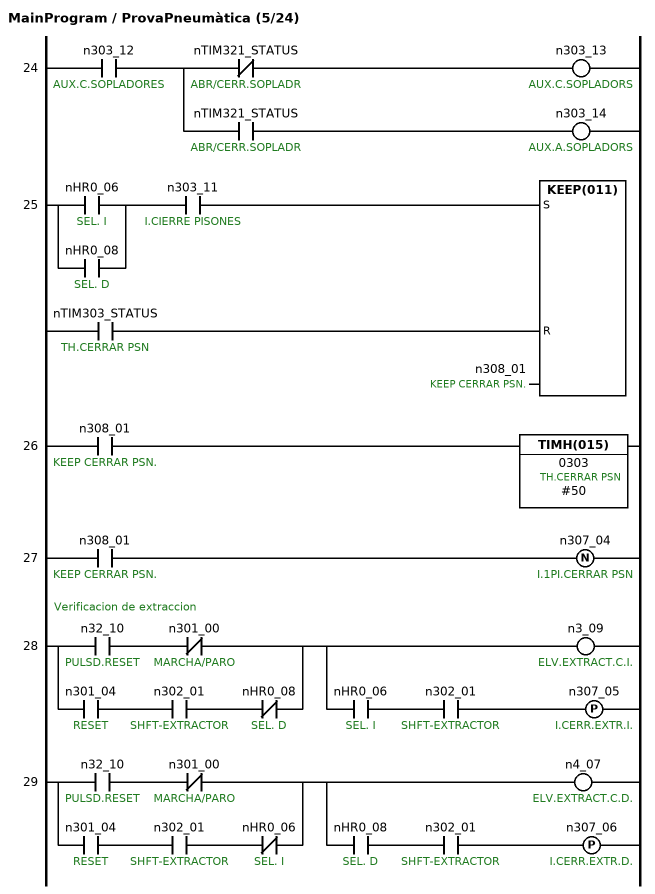
; [picture p96: MainProgram / ProvaPneumàtica, rungs 24-29]
; rung 24
LD n303_12  ; AUX.C.SOPLADORES
OUT TR0
ANDNOT nTIM321_STATUS  ; ABR/CERR.SOPLADR
OUT n303_13  ; AUX.C.SOPLADORS
LD TR0
AND nTIM321_STATUS  ; ABR/CERR.SOPLADR
OUT n303_14  ; AUX.A.SOPLADORS
; rung 25
LD nHR0_06  ; SEL. I
OR nHR0_08  ; SEL. D
AND n303_11  ; I.CIERRE PISONES
LD nTIM303_STATUS  ; TH.CERRAR PSN
KEEP(011) n308_01  ; KEEP CERRAR PSN.
; rung 26
LD n308_01  ; KEEP CERRAR PSN.
TIMH(015) 0303 #50  ; TH.CERRAR PSN
; rung 27
LD n308_01  ; KEEP CERRAR PSN.
DIFD(014) n307_04  ; I.1PI.CERRAR PSN
; rung 28: Verificacion de extraccion
LD n32_10  ; PULSD.RESET
ANDNOT n301_00  ; MARCHA/PARO
LD n301_04  ; RESET
AND n302_01  ; SHFT-EXTRACTOR
ANDNOT nHR0_08  ; SEL. D
ORLD
OUT n3_09  ; ELV.EXTRACT.C.I.
AND nHR0_06  ; SEL. I
AND n302_01  ; SHFT-EXTRACTOR
DIFU(013) n307_05  ; I.CERR.EXTR.I.
; rung 29
LD n32_10  ; PULSD.RESET
ANDNOT n301_00  ; MARCHA/PARO
LD n301_04  ; RESET
AND n302_01  ; SHFT-EXTRACTOR
ANDNOT nHR0_06  ; SEL. I
ORLD
OUT n4_07  ; ELV.EXTRACT.C.D.
AND nHR0_08  ; SEL. D
AND n302_01  ; SHFT-EXTRACTOR
DIFU(013) n307_06  ; I.CERR.EXTR.D.

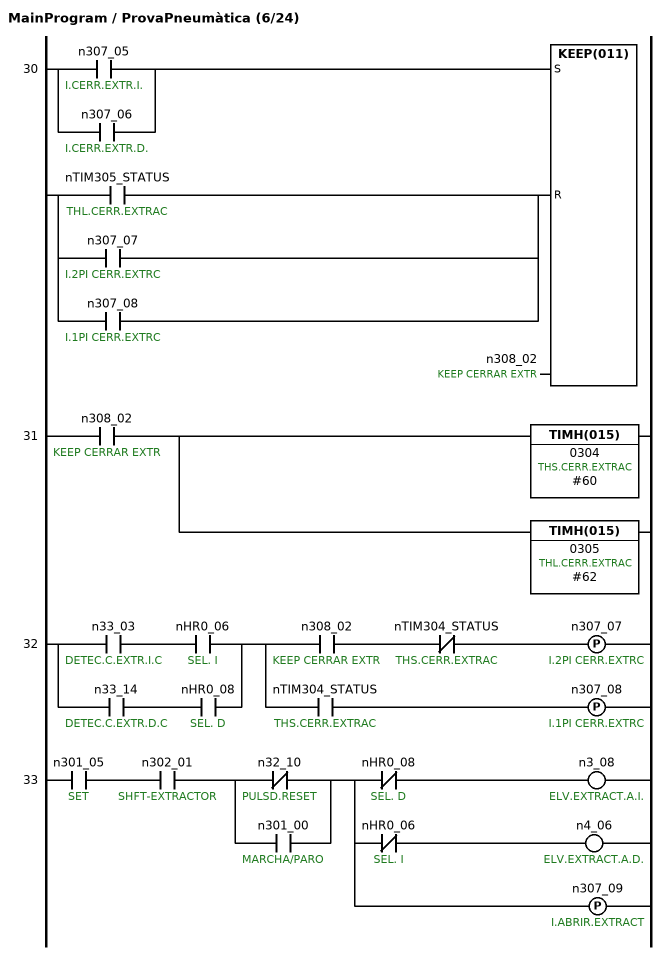
; rung 30
LD n307_05  ; I.CERR.EXTR.I.
OR n307_06  ; I.CERR.EXTR.D.
LD nTIM305_STATUS  ; THL.CERR.EXTRAC
OR n307_07  ; I.2PI CERR.EXTRC
OR n307_08  ; I.1PI CERR.EXTRC
KEEP(011) n308_02  ; KEEP CERRAR EXTR
; rung 31
LD n308_02  ; KEEP CERRAR EXTR
TIMH(015) 0304 #60  ; THS.CERR.EXTRAC
TIMH(015) 0305 #62  ; THL.CERR.EXTRAC
; rung 32
LD n33_03  ; DETEC.C.EXTR.I.C
AND nHR0_06  ; SEL. I
LD n33_14  ; DETEC.C.EXTR.D.C
AND nHR0_08  ; SEL. D
ORLD
OUT TR0
AND n308_02  ; KEEP CERRAR EXTR
ANDNOT nTIM304_STATUS  ; THS.CERR.EXTRAC
DIFU(013) n307_07  ; I.2PI CERR.EXTRC
LD TR0
AND nTIM304_STATUS  ; THS.CERR.EXTRAC
DIFU(013) n307_08  ; I.1PI CERR.EXTRC
; rung 33
LD n301_05  ; SET
AND n302_01  ; SHFT-EXTRACTOR
LDNOT n32_10  ; PULSD.RESET
OR n301_00  ; MARCHA/PARO
ANDLD
OUT TR0
ANDNOT nHR0_08  ; SEL. D
OUT n3_08  ; ELV.EXTRACT.A.I.
LD TR0
ANDNOT nHR0_06  ; SEL. I
OUT n4_06  ; ELV.EXTRACT.A.D.
LD TR0
DIFU(013) n307_09  ; I.ABRIR.EXTRACT

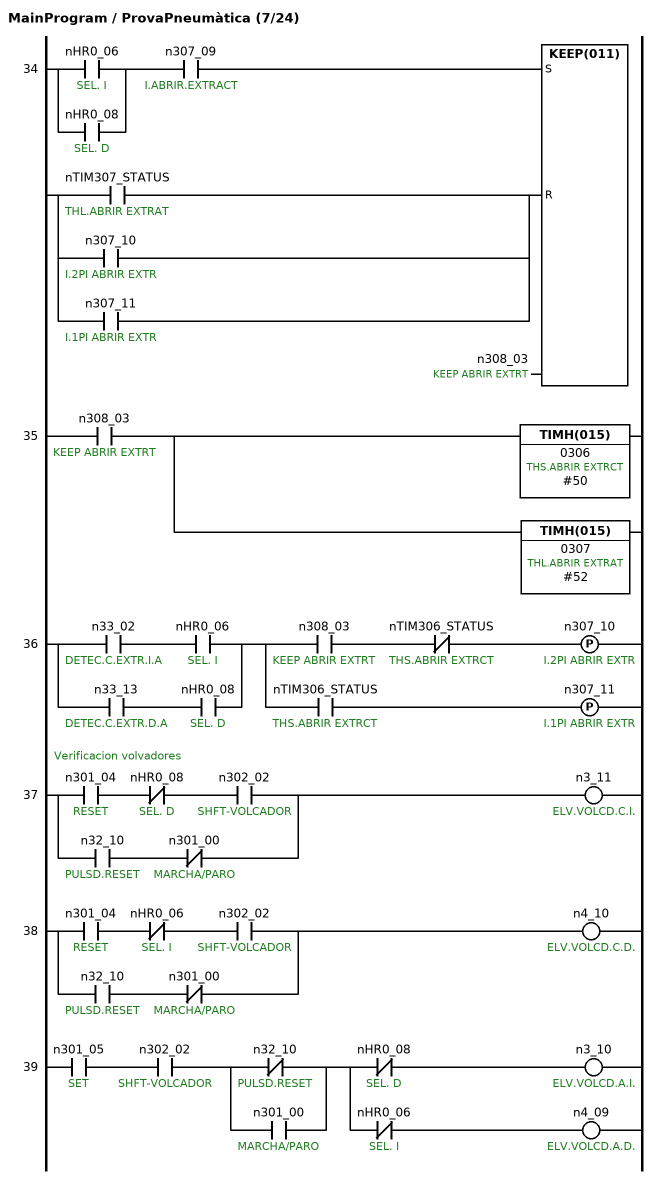
; rung 34
LD nHR0_06  ; SEL. I
OR nHR0_08  ; SEL. D
AND n307_09  ; I.ABRIR.EXTRACT
LD nTIM307_STATUS  ; THL.ABRIR EXTRAT
OR n307_10  ; I.2PI ABRIR EXTR
OR n307_11  ; I.1PI ABRIR EXTR
KEEP(011) n308_03  ; KEEP ABRIR EXTRT
; rung 35
LD n308_03  ; KEEP ABRIR EXTRT
TIMH(015) 0306 #50  ; THS.ABRIR EXTRCT
TIMH(015) 0307 #52  ; THL.ABRIR EXTRAT
; rung 36
LD n33_02  ; DETEC.C.EXTR.I.A
AND nHR0_06  ; SEL. I
LD n33_13  ; DETEC.C.EXTR.D.A
AND nHR0_08  ; SEL. D
ORLD
OUT TR0
AND n308_03  ; KEEP ABRIR EXTRT
ANDNOT nTIM306_STATUS  ; THS.ABRIR EXTRCT
DIFU(013) n307_10  ; I.2PI ABRIR EXTR
LD TR0
AND nTIM306_STATUS  ; THS.ABRIR EXTRCT
DIFU(013) n307_11  ; I.1PI ABRIR EXTR
; rung 37: Verificacion volvadores
LD n301_04  ; RESET
ANDNOT nHR0_08  ; SEL. D
AND n302_02  ; SHFT-VOLCADOR
LD n32_10  ; PULSD.RESET
ANDNOT n301_00  ; MARCHA/PARO
ORLD
OUT n3_11  ; ELV.VOLCD.C.I.
; rung 38
LD n301_04  ; RESET
ANDNOT nHR0_06  ; SEL. I
AND n302_02  ; SHFT-VOLCADOR
LD n32_10  ; PULSD.RESET
ANDNOT n301_00  ; MARCHA/PARO
ORLD
OUT n4_10  ; ELV.VOLCD.C.D.
; rung 39
LD n301_05  ; SET
AND n302_02  ; SHFT-VOLCADOR
LDNOT n32_10  ; PULSD.RESET
OR n301_00  ; MARCHA/PARO
ANDLD
OUT TR0
ANDNOT nHR0_08  ; SEL. D
OUT n3_10  ; ELV.VOLCD.A.I.
LD TR0
ANDNOT nHR0_06  ; SEL. I
OUT n4_09  ; ELV.VOLCD.A.D.

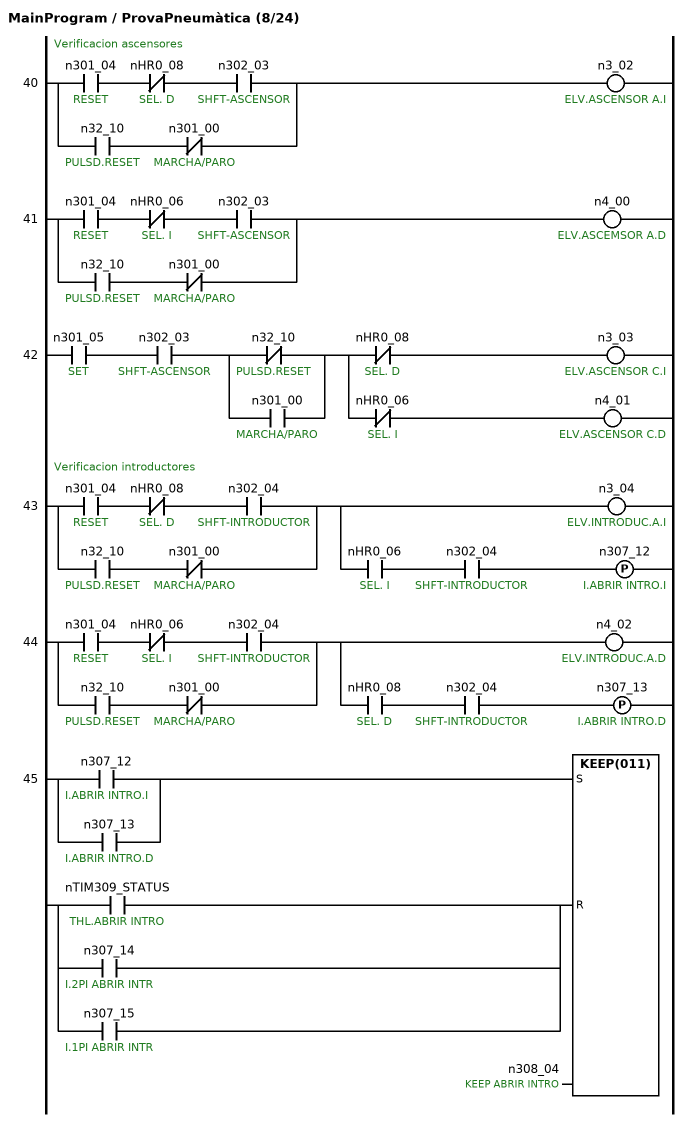
; rung 40: Verificacion ascensores
LD n301_04  ; RESET
ANDNOT nHR0_08  ; SEL. D
AND n302_03  ; SHFT-ASCENSOR
LD n32_10  ; PULSD.RESET
ANDNOT n301_00  ; MARCHA/PARO
ORLD
OUT n3_02  ; ELV.ASCENSOR A.I
; rung 41
LD n301_04  ; RESET
ANDNOT nHR0_06  ; SEL. I
AND n302_03  ; SHFT-ASCENSOR
LD n32_10  ; PULSD.RESET
ANDNOT n301_00  ; MARCHA/PARO
ORLD
OUT n4_00  ; ELV.ASCEMSOR A.D
; rung 42
LD n301_05  ; SET
AND n302_03  ; SHFT-ASCENSOR
LDNOT n32_10  ; PULSD.RESET
OR n301_00  ; MARCHA/PARO
ANDLD
OUT TR0
ANDNOT nHR0_08  ; SEL. D
OUT n3_03  ; ELV.ASCENSOR C.I
LD TR0
ANDNOT nHR0_06  ; SEL. I
OUT n4_01  ; ELV.ASCENSOR C.D
; rung 43: Verificacion introductores
LD n301_04  ; RESET
ANDNOT nHR0_08  ; SEL. D
AND n302_04  ; SHFT-INTRODUCTOR
LD n32_10  ; PULSD.RESET
ANDNOT n301_00  ; MARCHA/PARO
ORLD
OUT n3_04  ; ELV.INTRODUC.A.I
AND nHR0_06  ; SEL. I
AND n302_04  ; SHFT-INTRODUCTOR
DIFU(013) n307_12  ; I.ABRIR INTRO.I
; rung 44
LD n301_04  ; RESET
ANDNOT nHR0_06  ; SEL. I
AND n302_04  ; SHFT-INTRODUCTOR
LD n32_10  ; PULSD.RESET
ANDNOT n301_00  ; MARCHA/PARO
ORLD
OUT n4_02  ; ELV.INTRODUC.A.D
AND nHR0_08  ; SEL. D
AND n302_04  ; SHFT-INTRODUCTOR
DIFU(013) n307_13  ; I.ABRIR INTRO.D
; rung 45
LD n307_12  ; I.ABRIR INTRO.I
OR n307_13  ; I.ABRIR INTRO.D
LD nTIM309_STATUS  ; THL.ABRIR INTRO
OR n307_14  ; I.2PI ABRIR INTR
OR n307_15  ; I.1PI ABRIR INTR
KEEP(011) n308_04  ; KEEP ABRIR INTRO

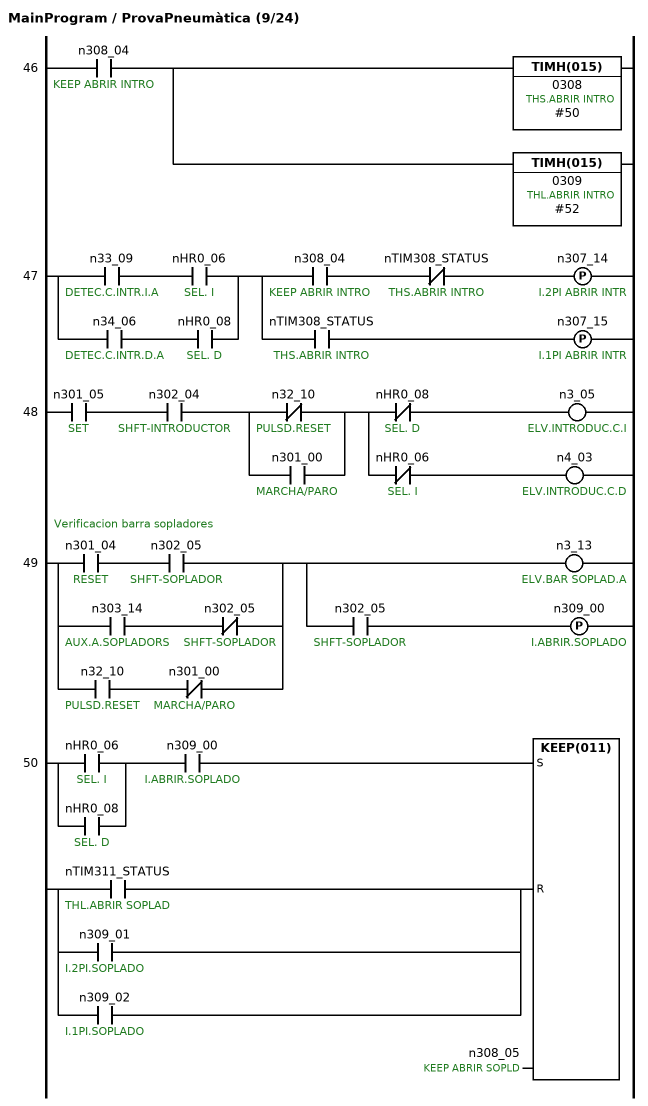
; rung 46
LD n308_04  ; KEEP ABRIR INTRO
TIMH(015) 0308 #50  ; THS.ABRIR INTRO
TIMH(015) 0309 #52  ; THL.ABRIR INTRO
; rung 47
LD n33_09  ; DETEC.C.INTR.I.A
AND nHR0_06  ; SEL. I
LD n34_06  ; DETEC.C.INTR.D.A
AND nHR0_08  ; SEL. D
ORLD
OUT TR0
AND n308_04  ; KEEP ABRIR INTRO
ANDNOT nTIM308_STATUS  ; THS.ABRIR INTRO
DIFU(013) n307_14  ; I.2PI ABRIR INTR
LD TR0
AND nTIM308_STATUS  ; THS.ABRIR INTRO
DIFU(013) n307_15  ; I.1PI ABRIR INTR
; rung 48
LD n301_05  ; SET
AND n302_04  ; SHFT-INTRODUCTOR
LDNOT n32_10  ; PULSD.RESET
OR n301_00  ; MARCHA/PARO
ANDLD
OUT TR0
ANDNOT nHR0_08  ; SEL. D
OUT n3_05  ; ELV.INTRODUC.C.I
LD TR0
ANDNOT nHR0_06  ; SEL. I
OUT n4_03  ; ELV.INTRODUC.C.D
; rung 49: Verificacion barra sopladores
LD n301_04  ; RESET
AND n302_05  ; SHFT-SOPLADOR
LD n303_14  ; AUX.A.SOPLADORS
ANDNOT n302_05  ; SHFT-SOPLADOR
ORLD
LD n32_10  ; PULSD.RESET
ANDNOT n301_00  ; MARCHA/PARO
ORLD
OUT n3_13  ; ELV.BAR SOPLAD.A
AND n302_05  ; SHFT-SOPLADOR
DIFU(013) n309_00  ; I.ABRIR.SOPLADO
; rung 50
LD nHR0_06  ; SEL. I
OR nHR0_08  ; SEL. D
AND n309_00  ; I.ABRIR.SOPLADO
LD nTIM311_STATUS  ; THL.ABRIR SOPLAD
OR n309_01  ; I.2PI.SOPLADO
OR n309_02  ; I.1PI.SOPLADO
KEEP(011) n308_05  ; KEEP ABRIR SOPLD

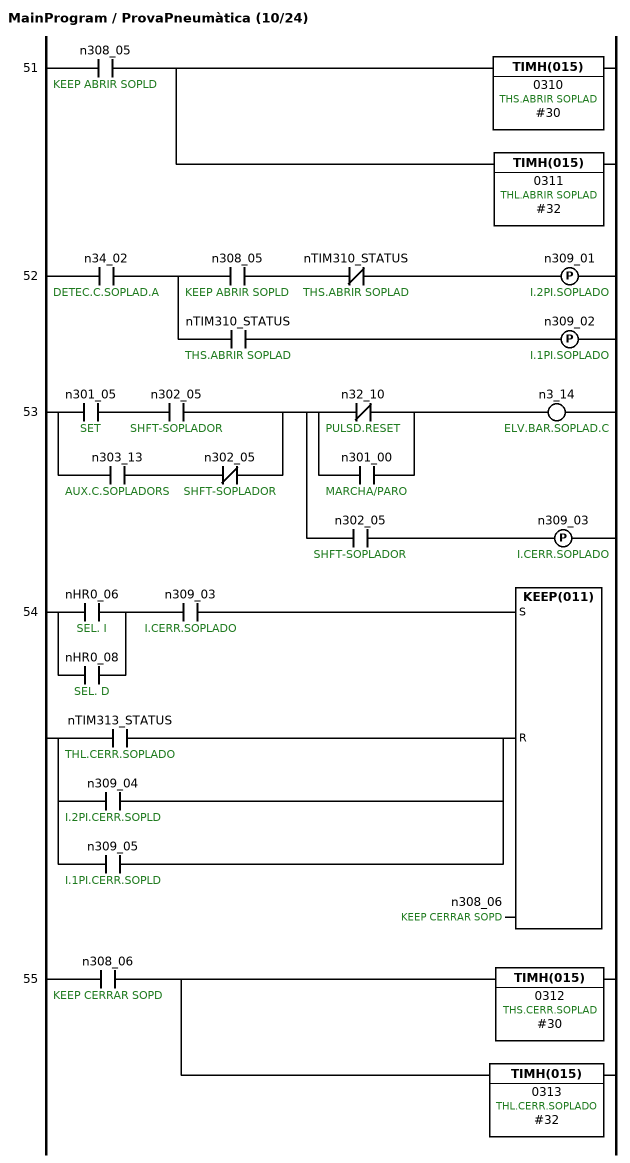
; rung 51
LD n308_05  ; KEEP ABRIR SOPLD
TIMH(015) 0310 #30  ; THS.ABRIR SOPLAD
TIMH(015) 0311 #32  ; THL.ABRIR SOPLAD
; rung 52
LD n34_02  ; DETEC.C.SOPLAD.A
OUT TR0
AND n308_05  ; KEEP ABRIR SOPLD
ANDNOT nTIM310_STATUS  ; THS.ABRIR SOPLAD
DIFU(013) n309_01  ; I.2PI.SOPLADO
LD TR0
AND nTIM310_STATUS  ; THS.ABRIR SOPLAD
DIFU(013) n309_02  ; I.1PI.SOPLADO
; rung 53
LD n301_05  ; SET
AND n302_05  ; SHFT-SOPLADOR
LD n303_13  ; AUX.C.SOPLADORS
ANDNOT n302_05  ; SHFT-SOPLADOR
ORLD
OUT TR0
LDNOT n32_10  ; PULSD.RESET
OR n301_00  ; MARCHA/PARO
ANDLD
OUT n3_14  ; ELV.BAR.SOPLAD.C
LD TR0
AND n302_05  ; SHFT-SOPLADOR
DIFU(013) n309_03  ; I.CERR.SOPLADO
; rung 54
LD nHR0_06  ; SEL. I
OR nHR0_08  ; SEL. D
AND n309_03  ; I.CERR.SOPLADO
LD nTIM313_STATUS  ; THL.CERR.SOPLADO
OR n309_04  ; I.2PI.CERR.SOPLD
OR n309_05  ; I.1PI.CERR.SOPLD
KEEP(011) n308_06  ; KEEP CERRAR SOPD
; rung 55
LD n308_06  ; KEEP CERRAR SOPD
TIMH(015) 0312 #30  ; THS.CERR.SOPLAD
TIMH(015) 0313 #32  ; THL.CERR.SOPLADO

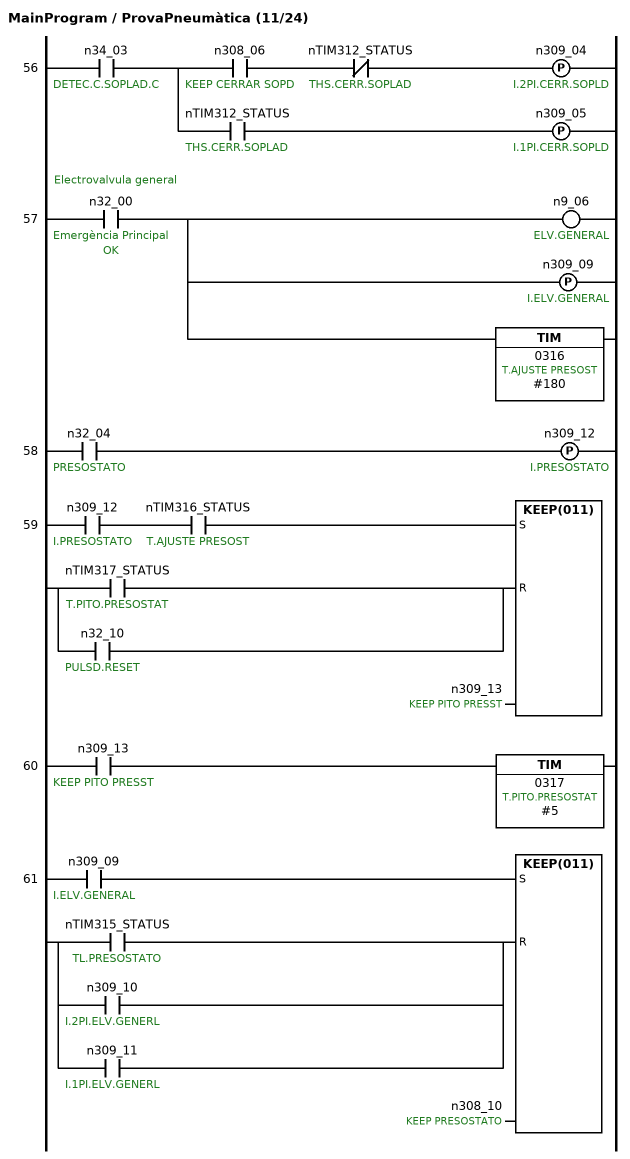
; rung 56
LD n34_03  ; DETEC.C.SOPLAD.C
OUT TR0
AND n308_06  ; KEEP CERRAR SOPD
ANDNOT nTIM312_STATUS  ; THS.CERR.SOPLAD
DIFU(013) n309_04  ; I.2PI.CERR.SOPLD
LD TR0
AND nTIM312_STATUS  ; THS.CERR.SOPLAD
DIFU(013) n309_05  ; I.1PI.CERR.SOPLD
; rung 57: Electrovalvula general
LD n32_00  ; Emergència Principal OK
OUT n9_06  ; ELV.GENERAL
DIFU(013) n309_09  ; I.ELV.GENERAL
TIM 0316 #180  ; T.AJUSTE PRESOST
; rung 58
LD n32_04  ; PRESOSTATO
DIFU(013) n309_12  ; I.PRESOSTATO
; rung 59
LD n309_12  ; I.PRESOSTATO
AND nTIM316_STATUS  ; T.AJUSTE PRESOST
LD nTIM317_STATUS  ; T.PITO.PRESOSTAT
OR n32_10  ; PULSD.RESET
KEEP(011) n309_13  ; KEEP PITO PRESST
; rung 60
LD n309_13  ; KEEP PITO PRESST
TIM 0317 #5  ; T.PITO.PRESOSTAT
; rung 61
LD n309_09  ; I.ELV.GENERAL
LD nTIM315_STATUS  ; TL.PRESOSTATO
OR n309_10  ; I.2PI.ELV.GENERL
OR n309_11  ; I.1PI.ELV.GENERL
KEEP(011) n308_10  ; KEEP PRESOSTATO

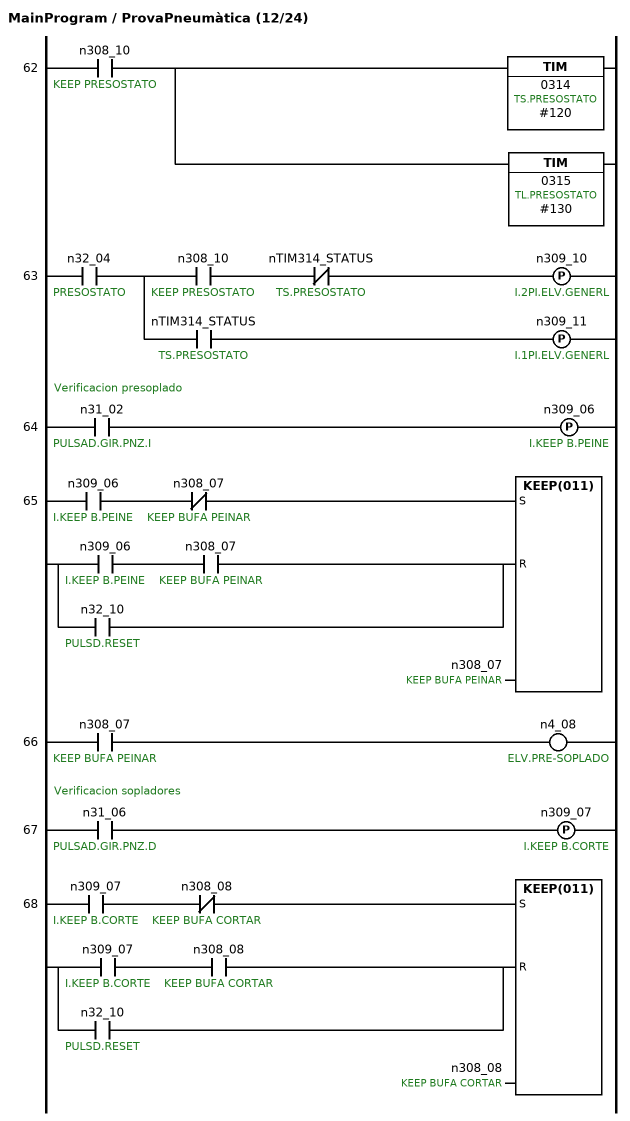
; rung 62
LD n308_10  ; KEEP PRESOSTATO
TIM 0314 #120  ; TS.PRESOSTATO
TIM 0315 #130  ; TL.PRESOSTATO
; rung 63
LD n32_04  ; PRESOSTATO
OUT TR0
AND n308_10  ; KEEP PRESOSTATO
ANDNOT nTIM314_STATUS  ; TS.PRESOSTATO
DIFU(013) n309_10  ; I.2PI.ELV.GENERL
LD TR0
AND nTIM314_STATUS  ; TS.PRESOSTATO
DIFU(013) n309_11  ; I.1PI.ELV.GENERL
; rung 64: Verificacion presoplado
LD n31_02  ; PULSAD.GIR.PNZ.I
DIFU(013) n309_06  ; I.KEEP B.PEINE
; rung 65
LD n309_06  ; I.KEEP B.PEINE
ANDNOT n308_07  ; KEEP BUFA PEINAR
LD n309_06  ; I.KEEP B.PEINE
AND n308_07  ; KEEP BUFA PEINAR
OR n32_10  ; PULSD.RESET
KEEP(011) n308_07  ; KEEP BUFA PEINAR
; rung 66
LD n308_07  ; KEEP BUFA PEINAR
OUT n4_08  ; ELV.PRE-SOPLADO
; rung 67: Verificacion sopladores
LD n31_06  ; PULSAD.GIR.PNZ.D
DIFU(013) n309_07  ; I.KEEP B.CORTE
; rung 68
LD n309_07  ; I.KEEP B.CORTE
ANDNOT n308_08  ; KEEP BUFA CORTAR
LD n309_07  ; I.KEEP B.CORTE
AND n308_08  ; KEEP BUFA CORTAR
OR n32_10  ; PULSD.RESET
KEEP(011) n308_08  ; KEEP BUFA CORTAR

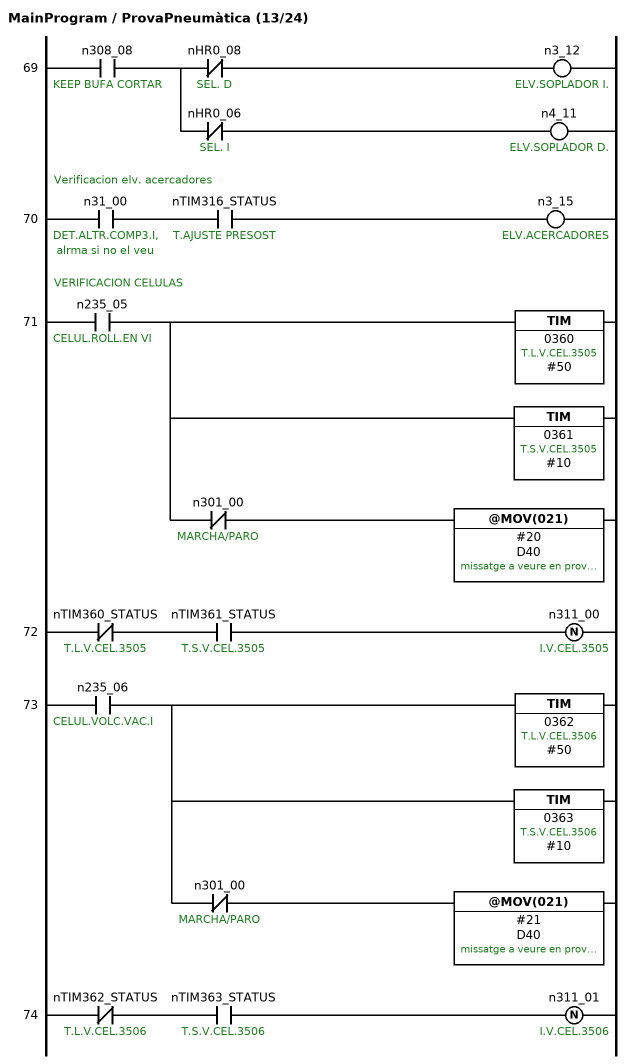
; rung 69
LD n308_08  ; KEEP BUFA CORTAR
OUT TR0
ANDNOT nHR0_08  ; SEL. D
OUT n3_12  ; ELV.SOPLADOR I.
LD TR0
ANDNOT nHR0_06  ; SEL. I
OUT n4_11  ; ELV.SOPLADOR D.
; rung 70: Verificacion elv. acercadores
LD n31_00  ; DET.ALTR.COMP3.I, alrma si no el veu
AND nTIM316_STATUS  ; T.AJUSTE PRESOST
OUT n3_15  ; ELV.ACERCADORES
; rung 71: VERIFICACION CELULAS
LD n235_05  ; CELUL.ROLL.EN VI
TIM 0360 #50  ; T.L.V.CEL.3505
TIM 0361 #10  ; T.S.V.CEL.3505
ANDNOT n301_00  ; MARCHA/PARO
@MOV(021) #20 D40  ; missatge a veure en prova pneumàtica
; rung 72
LDNOT nTIM360_STATUS  ; T.L.V.CEL.3505
AND nTIM361_STATUS  ; T.S.V.CEL.3505
DIFD(014) n311_00  ; I.V.CEL.3505
; rung 73
LD n235_06  ; CELUL.VOLC.VAC.I
TIM 0362 #50  ; T.L.V.CEL.3506
TIM 0363 #10  ; T.S.V.CEL.3506
ANDNOT n301_00  ; MARCHA/PARO
@MOV(021) #21 D40  ; missatge a veure en prova pneumàtica
; rung 74
LDNOT nTIM362_STATUS  ; T.L.V.CEL.3506
AND nTIM363_STATUS  ; T.S.V.CEL.3506
DIFD(014) n311_01  ; I.V.CEL.3506

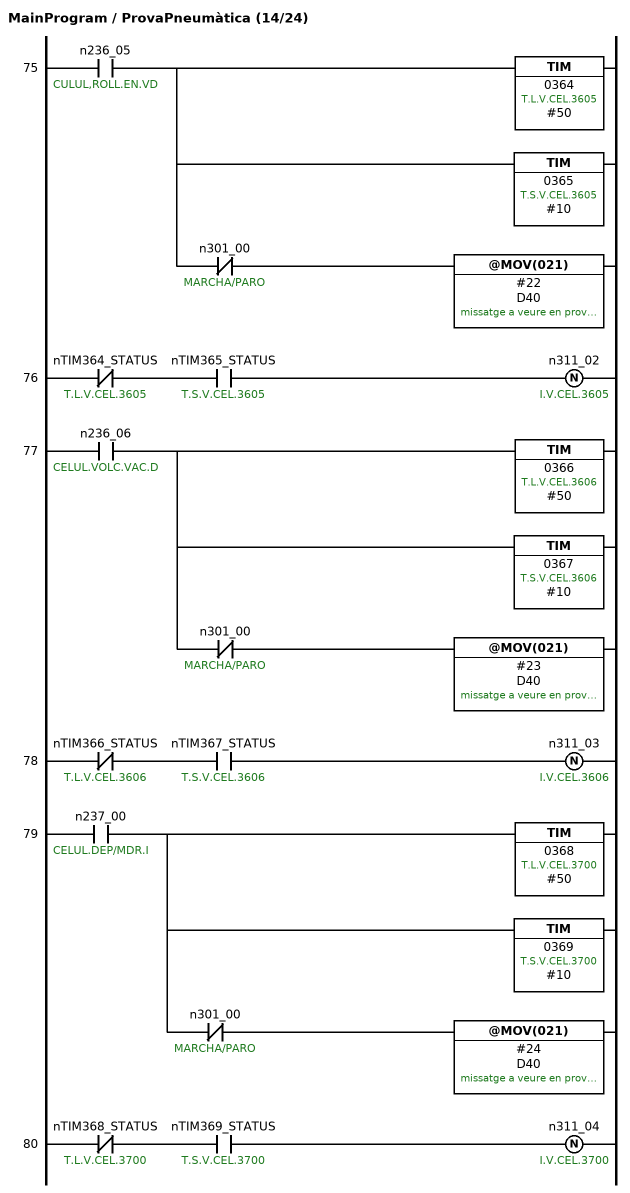
; rung 75
LD n236_05  ; CULUL,ROLL.EN.VD
TIM 0364 #50  ; T.L.V.CEL.3605
TIM 0365 #10  ; T.S.V.CEL.3605
ANDNOT n301_00  ; MARCHA/PARO
@MOV(021) #22 D40  ; missatge a veure en prova pneumàtica
; rung 76
LDNOT nTIM364_STATUS  ; T.L.V.CEL.3605
AND nTIM365_STATUS  ; T.S.V.CEL.3605
DIFD(014) n311_02  ; I.V.CEL.3605
; rung 77
LD n236_06  ; CELUL.VOLC.VAC.D
TIM 0366 #50  ; T.L.V.CEL.3606
TIM 0367 #10  ; T.S.V.CEL.3606
ANDNOT n301_00  ; MARCHA/PARO
@MOV(021) #23 D40  ; missatge a veure en prova pneumàtica
; rung 78
LDNOT nTIM366_STATUS  ; T.L.V.CEL.3606
AND nTIM367_STATUS  ; T.S.V.CEL.3606
DIFD(014) n311_03  ; I.V.CEL.3606
; rung 79
LD n237_00  ; CELUL.DEP/MDR.I
TIM 0368 #50  ; T.L.V.CEL.3700
TIM 0369 #10  ; T.S.V.CEL.3700
ANDNOT n301_00  ; MARCHA/PARO
@MOV(021) #24 D40  ; missatge a veure en prova pneumàtica
; rung 80
LDNOT nTIM368_STATUS  ; T.L.V.CEL.3700
AND nTIM369_STATUS  ; T.S.V.CEL.3700
DIFD(014) n311_04  ; I.V.CEL.3700

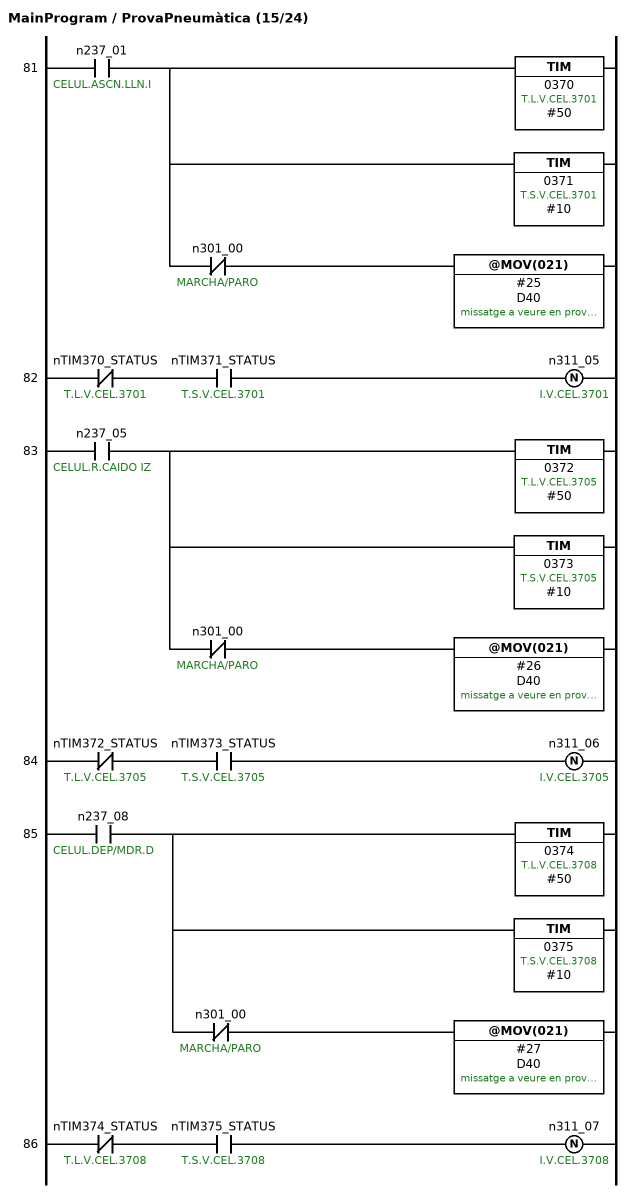
; rung 81
LD n237_01  ; CELUL.ASCN.LLN.I
TIM 0370 #50  ; T.L.V.CEL.3701
TIM 0371 #10  ; T.S.V.CEL.3701
ANDNOT n301_00  ; MARCHA/PARO
@MOV(021) #25 D40  ; missatge a veure en prova pneumàtica
; rung 82
LDNOT nTIM370_STATUS  ; T.L.V.CEL.3701
AND nTIM371_STATUS  ; T.S.V.CEL.3701
DIFD(014) n311_05  ; I.V.CEL.3701
; rung 83
LD n237_05  ; CELUL.R.CAIDO IZ
TIM 0372 #50  ; T.L.V.CEL.3705
TIM 0373 #10  ; T.S.V.CEL.3705
ANDNOT n301_00  ; MARCHA/PARO
@MOV(021) #26 D40  ; missatge a veure en prova pneumàtica
; rung 84
LDNOT nTIM372_STATUS  ; T.L.V.CEL.3705
AND nTIM373_STATUS  ; T.S.V.CEL.3705
DIFD(014) n311_06  ; I.V.CEL.3705
; rung 85
LD n237_08  ; CELUL.DEP/MDR.D
TIM 0374 #50  ; T.L.V.CEL.3708
TIM 0375 #10  ; T.S.V.CEL.3708
ANDNOT n301_00  ; MARCHA/PARO
@MOV(021) #27 D40  ; missatge a veure en prova pneumàtica
; rung 86
LDNOT nTIM374_STATUS  ; T.L.V.CEL.3708
AND nTIM375_STATUS  ; T.S.V.CEL.3708
DIFD(014) n311_07  ; I.V.CEL.3708

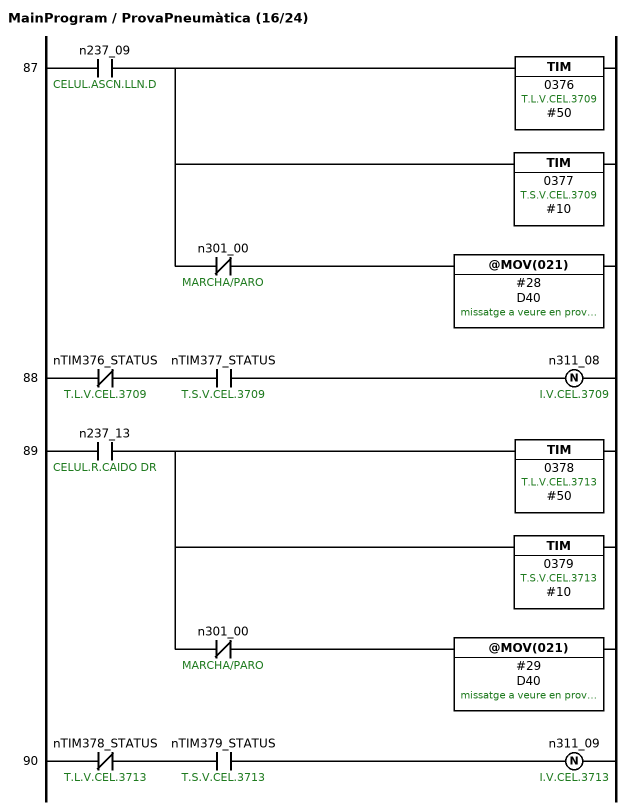
; rung 87
LD n237_09  ; CELUL.ASCN.LLN.D
TIM 0376 #50  ; T.L.V.CEL.3709
TIM 0377 #10  ; T.S.V.CEL.3709
ANDNOT n301_00  ; MARCHA/PARO
@MOV(021) #28 D40  ; missatge a veure en prova pneumàtica
; rung 88
LDNOT nTIM376_STATUS  ; T.L.V.CEL.3709
AND nTIM377_STATUS  ; T.S.V.CEL.3709
DIFD(014) n311_08  ; I.V.CEL.3709
; rung 89
LD n237_13  ; CELUL.R.CAIDO DR
TIM 0378 #50  ; T.L.V.CEL.3713
TIM 0379 #10  ; T.S.V.CEL.3713
ANDNOT n301_00  ; MARCHA/PARO
@MOV(021) #29 D40  ; missatge a veure en prova pneumàtica
; rung 90
LDNOT nTIM378_STATUS  ; T.L.V.CEL.3713
AND nTIM379_STATUS  ; T.S.V.CEL.3713
DIFD(014) n311_09  ; I.V.CEL.3713

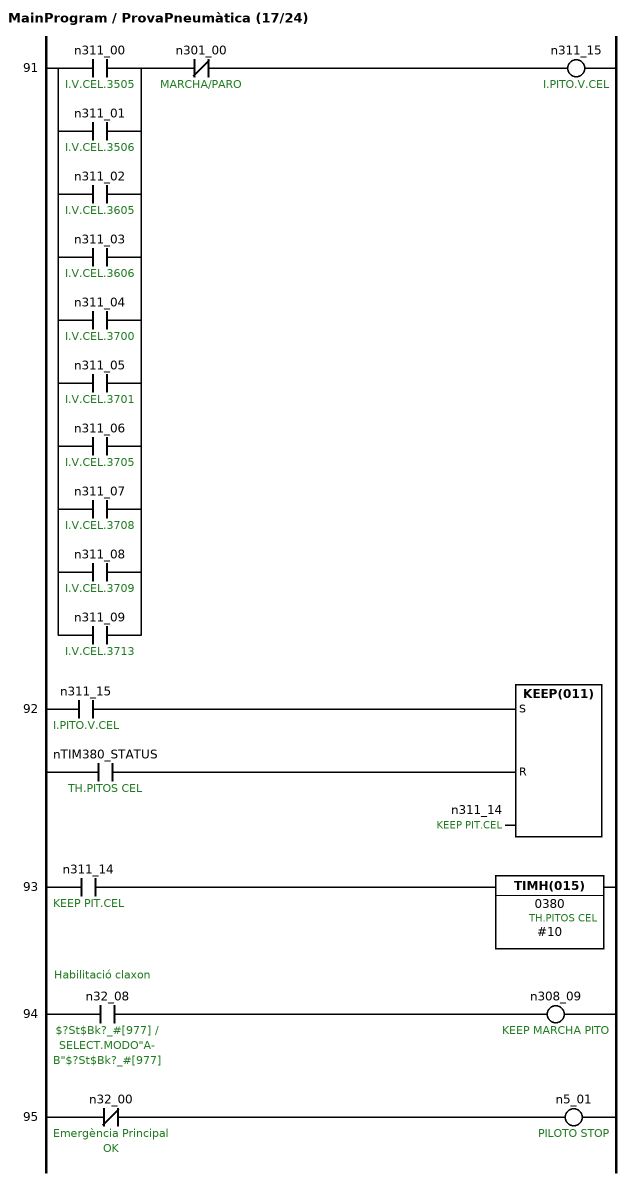
; rung 91
LD n311_00  ; I.V.CEL.3505
OR n311_01  ; I.V.CEL.3506
OR n311_02  ; I.V.CEL.3605
OR n311_03  ; I.V.CEL.3606
OR n311_04  ; I.V.CEL.3700
OR n311_05  ; I.V.CEL.3701
OR n311_06  ; I.V.CEL.3705
OR n311_07  ; I.V.CEL.3708
OR n311_08  ; I.V.CEL.3709
OR n311_09  ; I.V.CEL.3713
ANDNOT n301_00  ; MARCHA/PARO
OUT n311_15  ; I.PITO.V.CEL
; rung 92
LD n311_15  ; I.PITO.V.CEL
LD nTIM380_STATUS  ; TH.PITOS CEL
KEEP(011) n311_14  ; KEEP PIT.CEL
; rung 93
LD n311_14  ; KEEP PIT.CEL
TIMH(015) 0380 #10  ; TH.PITOS CEL
; rung 94: Habilitació claxon
LD n32_08  ; $?St$Bk?_#[977] / SELECT.MODO"A-B"$?St$Bk?_#[977]
OUT n308_09  ; KEEP MARCHA PITO
; rung 95
LDNOT n32_00  ; Emergència Principal OK
OUT n5_01  ; PILOTO STOP

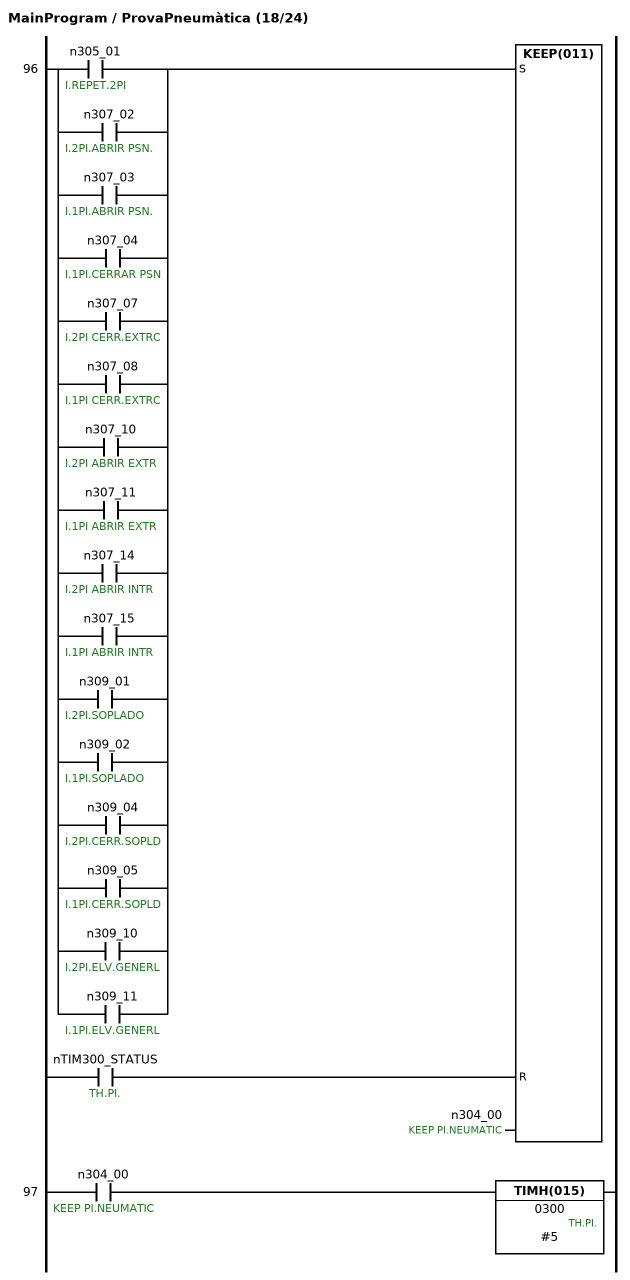
; rung 96
LD n305_01  ; I.REPET.2PI
OR n307_02  ; I.2PI.ABRIR PSN.
OR n307_03  ; I.1PI.ABRIR PSN.
OR n307_04  ; I.1PI.CERRAR PSN
OR n307_07  ; I.2PI CERR.EXTRC
OR n307_08  ; I.1PI CERR.EXTRC
OR n307_10  ; I.2PI ABRIR EXTR
OR n307_11  ; I.1PI ABRIR EXTR
OR n307_14  ; I.2PI ABRIR INTR
OR n307_15  ; I.1PI ABRIR INTR
OR n309_01  ; I.2PI.SOPLADO
OR n309_02  ; I.1PI.SOPLADO
OR n309_04  ; I.2PI.CERR.SOPLD
OR n309_05  ; I.1PI.CERR.SOPLD
OR n309_10  ; I.2PI.ELV.GENERL
OR n309_11  ; I.1PI.ELV.GENERL
LD nTIM300_STATUS  ; TH.PI.
KEEP(011) n304_00  ; KEEP PI.NEUMATIC
; rung 97
LD n304_00  ; KEEP PI.NEUMATIC
TIMH(015) 0300 #5  ; TH.PI.

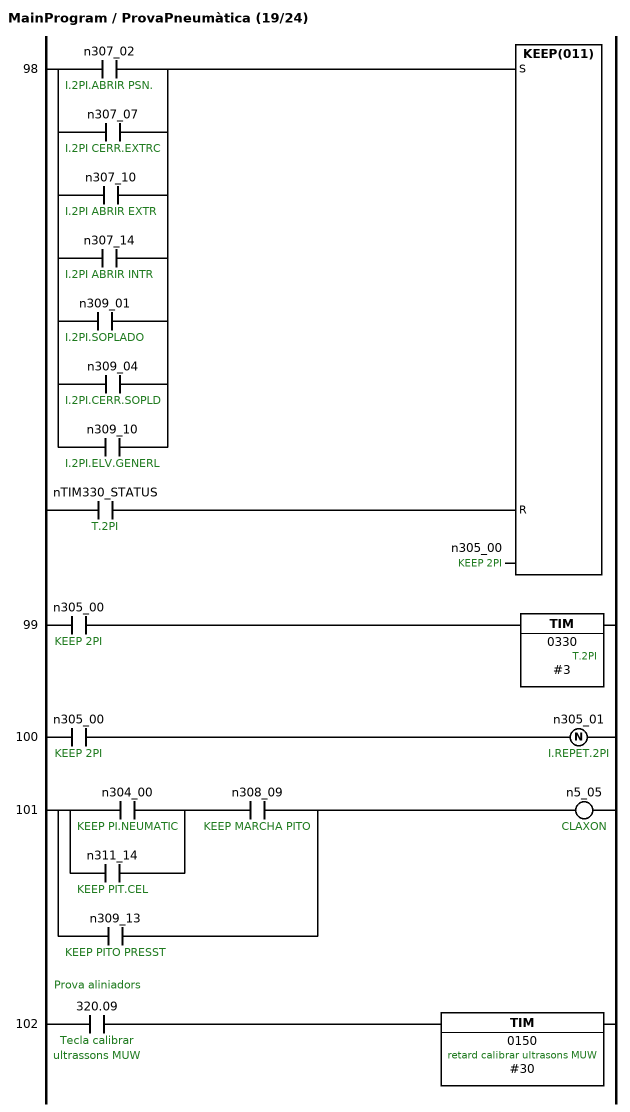
; rung 98
LD n307_02  ; I.2PI.ABRIR PSN.
OR n307_07  ; I.2PI CERR.EXTRC
OR n307_10  ; I.2PI ABRIR EXTR
OR n307_14  ; I.2PI ABRIR INTR
OR n309_01  ; I.2PI.SOPLADO
OR n309_04  ; I.2PI.CERR.SOPLD
OR n309_10  ; I.2PI.ELV.GENERL
LD nTIM330_STATUS  ; T.2PI
KEEP(011) n305_00  ; KEEP 2PI
; rung 99
LD n305_00  ; KEEP 2PI
TIM 0330 #3  ; T.2PI
; rung 100
LD n305_00  ; KEEP 2PI
DIFD(014) n305_01  ; I.REPET.2PI
; rung 101
LD n304_00  ; KEEP PI.NEUMATIC
OR n311_14  ; KEEP PIT.CEL
AND n308_09  ; KEEP MARCHA PITO
OR n309_13  ; KEEP PITO PRESST
OUT n5_05  ; CLAXON
; rung 102: Prova aliniadors
LD 320.09  ; Tecla calibrar ultrassons MUW
TIM 0150 #30  ; retard calibrar ultrasons MUW

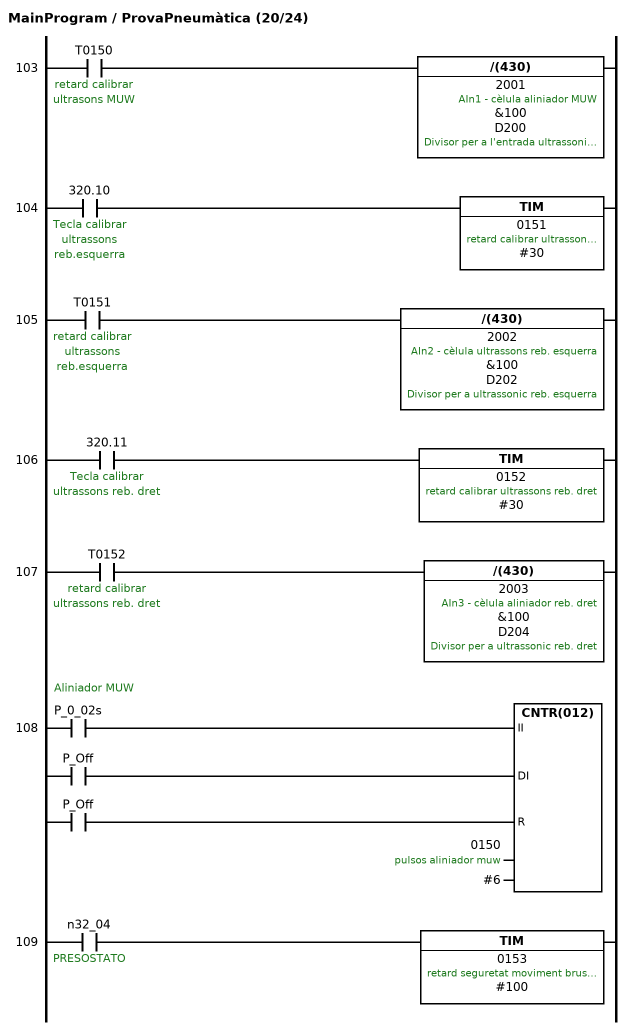
; rung 103
LD T0150  ; retard calibrar ultrasons MUW
/(430) 2001 &100 D200  ; AIn1 - cèlula aliniador MUW, Divisor per a l'entrada ultrassonic MUW
; rung 104
LD 320.10  ; Tecla calibrar ultrassons reb.esquerra
TIM 0151 #30  ; retard calibrar ultrassons reb.esquerra
; rung 105
LD T0151  ; retard calibrar ultrassons reb.esquerra
/(430) 2002 &100 D202  ; AIn2 - cèlula ultrassons reb. esquerra, Divisor per a ultrassonic reb. esquerra
; rung 106
LD 320.11  ; Tecla calibrar ultrassons reb. dret
TIM 0152 #30  ; retard calibrar ultrassons reb. dret
; rung 107
LD T0152  ; retard calibrar ultrassons reb. dret
/(430) 2003 &100 D204  ; AIn3 - cèlula aliniador reb. dret, Divisor per a ultrassonic reb. dret
; rung 108: Aliniador MUW
LD P_0_02s
LD P_Off
LD P_Off
CNTR(012) 0150 #6  ; pulsos aliniador muw
; rung 109
LD n32_04  ; PRESOSTATO
TIM 0153 #100  ; retard seguretat moviment brusc aliniador MUW

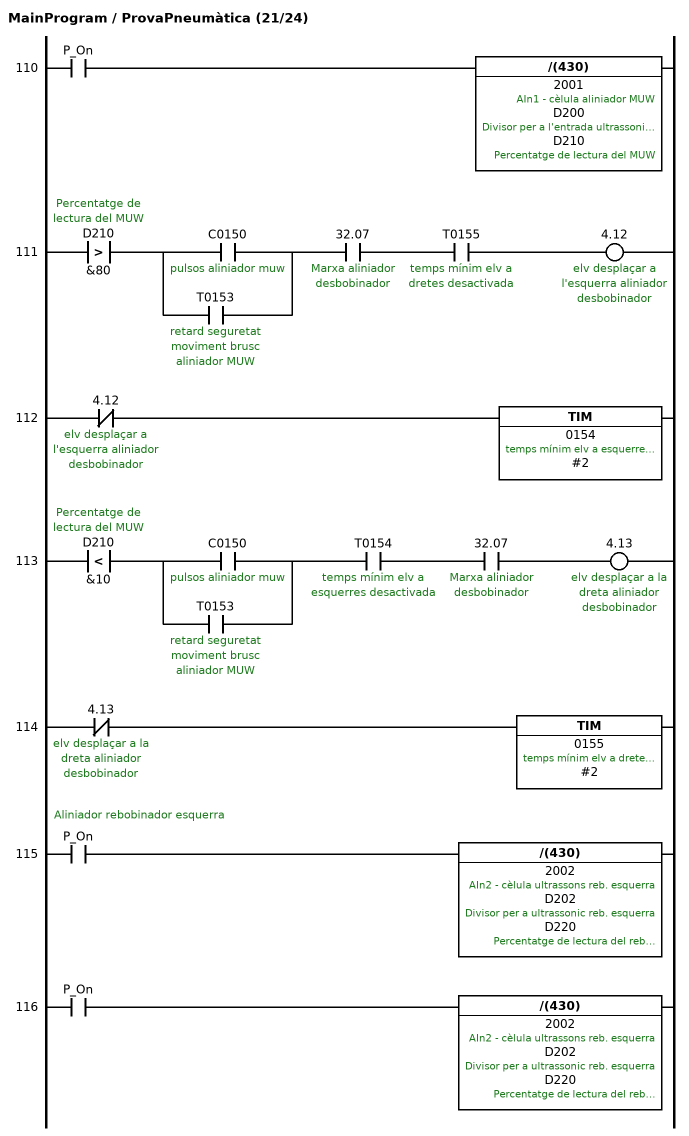
; rung 110
LD P_On
/(430) 2001 D200 D210  ; AIn1 - cèlula aliniador MUW, Divisor per a l'entrada ultrassonic MUW, Percentatge de lectura del MUW
; rung 111
LD>(320) D210 &80  ; Percentatge de lectura del MUW
LD C0150  ; pulsos aliniador muw
OR T0153  ; retard seguretat moviment brusc aliniador MUW
ANDLD
AND 32.07  ; Marxa aliniador desbobinador
AND T0155  ; temps mínim elv a dretes desactivada
OUT 4.12  ; elv desplaçar a l'esquerra aliniador desbobinador
; rung 112
LDNOT 4.12  ; elv desplaçar a l'esquerra aliniador desbobinador
TIM 0154 #2  ; temps mínim elv a esquerres desactivada
; rung 113
LD<(310) D210 &10  ; Percentatge de lectura del MUW
LD C0150  ; pulsos aliniador muw
OR T0153  ; retard seguretat moviment brusc aliniador MUW
ANDLD
AND T0154  ; temps mínim elv a esquerres desactivada
AND 32.07  ; Marxa aliniador desbobinador
OUT 4.13  ; elv desplaçar a la dreta aliniador desbobinador
; rung 114
LDNOT 4.13  ; elv desplaçar a la dreta aliniador desbobinador
TIM 0155 #2  ; temps mínim elv a dretes desactivada
; rung 115: Aliniador rebobinador esquerra
LD P_On
/(430) 2002 D202 D220  ; AIn2 - cèlula ultrassons reb. esquerra, Divisor per a ultrassonic reb. esquerra, Percentatge de lectura del reb. esquerra
; rung 116
LD P_On
/(430) 2002 D202 D220  ; AIn2 - cèlula ultrassons reb. esquerra, Divisor per a ultrassonic reb. esquerra, Percentatge de lectura del reb. esquerra

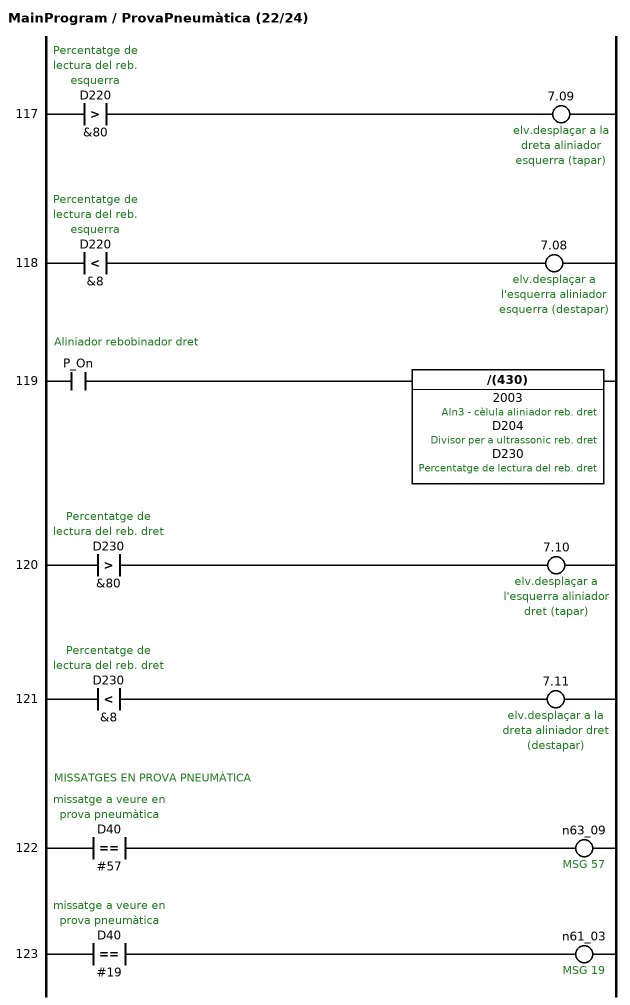
; rung 117
LD>(320) D220 &80  ; Percentatge de lectura del reb. esquerra
OUT 7.09  ; elv.desplaçar a la dreta aliniador esquerra (tapar)
; rung 118
LD<(310) D220 &8  ; Percentatge de lectura del reb. esquerra
OUT 7.08  ; elv.desplaçar a l'esquerra aliniador esquerra (destapar)
; rung 119: Aliniador rebobinador dret
LD P_On
/(430) 2003 D204 D230  ; AIn3 - cèlula aliniador reb. dret, Divisor per a ultrassonic reb. dret, Percentatge de lectura del reb. dret
; rung 120
LD>(320) D230 &80  ; Percentatge de lectura del reb. dret
OUT 7.10  ; elv.desplaçar a l'esquerra aliniador dret (tapar)
; rung 121
LD<(310) D230 &8  ; Percentatge de lectura del reb. dret
OUT 7.11  ; elv.desplaçar a la dreta aliniador dret (destapar)
; rung 122: MISSATGES EN PROVA PNEUMÀTICA
LD=(300) D40 #57  ; missatge a veure en prova pneumàtica
OUT n63_09  ; MSG 57
; rung 123
LD=(300) D40 #19  ; missatge a veure en prova pneumàtica
OUT n61_03  ; MSG 19

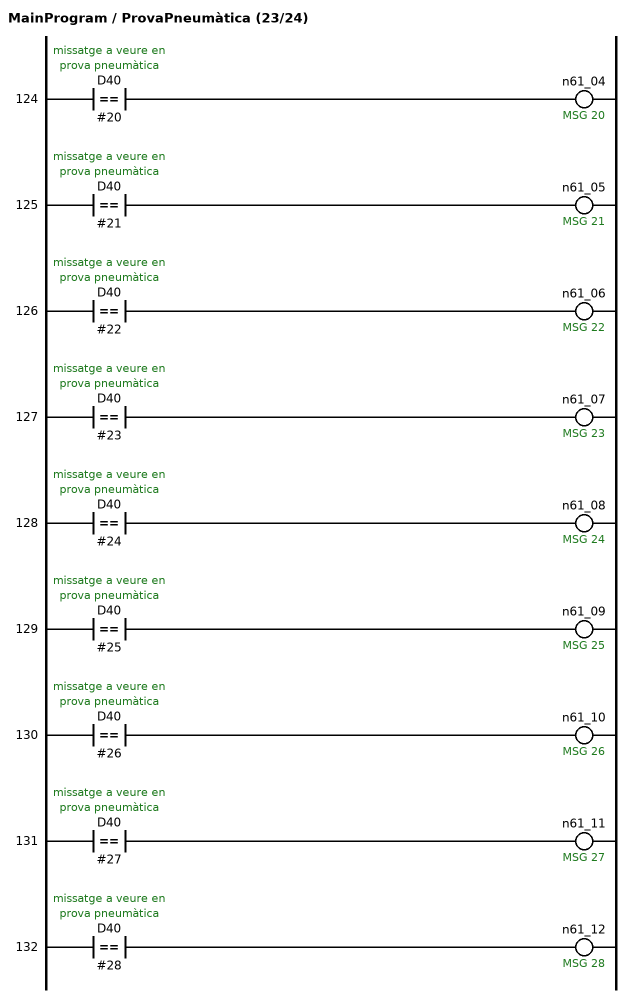
; rung 124
LD=(300) D40 #20  ; missatge a veure en prova pneumàtica
OUT n61_04  ; MSG 20
; rung 125
LD=(300) D40 #21  ; missatge a veure en prova pneumàtica
OUT n61_05  ; MSG 21
; rung 126
LD=(300) D40 #22  ; missatge a veure en prova pneumàtica
OUT n61_06  ; MSG 22
; rung 127
LD=(300) D40 #23  ; missatge a veure en prova pneumàtica
OUT n61_07  ; MSG 23
; rung 128
LD=(300) D40 #24  ; missatge a veure en prova pneumàtica
OUT n61_08  ; MSG 24
; rung 129
LD=(300) D40 #25  ; missatge a veure en prova pneumàtica
OUT n61_09  ; MSG 25
; rung 130
LD=(300) D40 #26  ; missatge a veure en prova pneumàtica
OUT n61_10  ; MSG 26
; rung 131
LD=(300) D40 #27  ; missatge a veure en prova pneumàtica
OUT n61_11  ; MSG 27
; rung 132
LD=(300) D40 #28  ; missatge a veure en prova pneumàtica
OUT n61_12  ; MSG 28

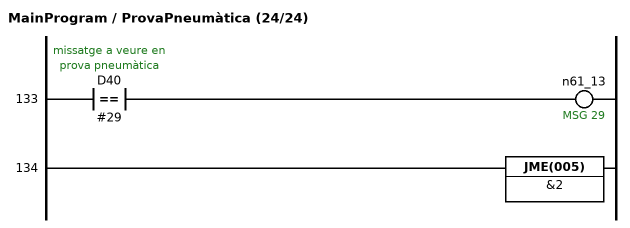
; rung 133
LD=(300) D40 #29  ; missatge a veure en prova pneumàtica
OUT n61_13  ; MSG 29
; rung 134
JME(005) &2
; rung 135: LAS DENOMINACIONES ELV.A. Y ELV.C SE ENTIENDEN RESPECTO AL / MOVIMIENTO DE SU PISTON CORRESPONDIENTE Y NO AL ELEMENTO.

### Section END
; rung 0
END(001)